// TIA Portal V19 export
TYPE "MatCountPersistent"
// stored: Access Published
   STRUCT
      Data : "MatCountData";
      Par { S7_SetPoint := 'True'} : "MatCountPar";
   END_STRUCT;
END_TYPE
